SUBAPPLICATION Uebung_016a (* Background Colour umschalten -- 3-fach *)
  (* Standard: 61499-2; Description: Copyright (c) 2023 Meisterschulen am Ostbahnhof This program and the accompanying materials are made available under the terms of the Eclipse Public License 2.0 which is available at https://www.eclipse.org/legal/epl-2.0/ SPDX-License-Identifier: EPL-2.0 *)
  (* Version 1.0, 2023-10-23, Franz Höpfinger, Meisterschulen am Ostbahnhof *)
  IMPORT DefaultPool::SoftKey_F1;
  IMPORT DefaultPool::SoftKey_F2;
  IMPORT DefaultPool::SoftKey_F3;
  IMPORT DefaultPool::SoftKey_F7;
  IMPORT SoftKeyActivationCode::SK_RELEASED;
  IMPORT isobus::ut::colours::COLOR_GREEN;
  IMPORT isobus::ut::colours::COLOR_RED;
  IMPORT isobus::ut::colours::COLOR_WHITE;
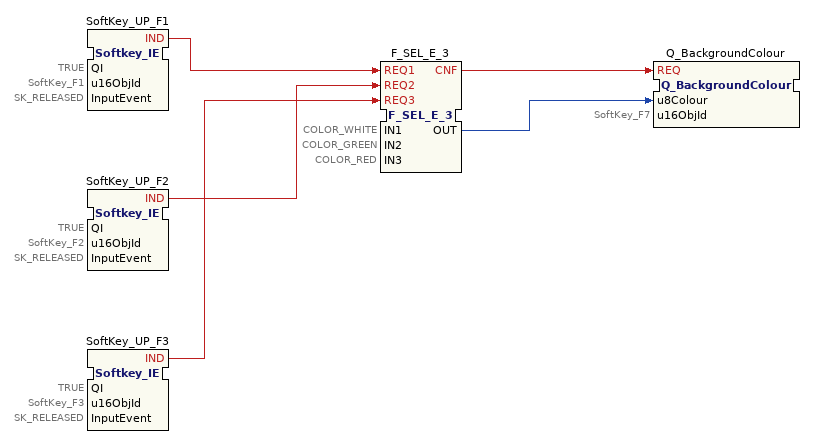
  FBS
    SoftKey_UP_F1 : Softkey_IE(QI := TRUE, u16ObjId := SoftKey_F1, InputEvent := SK_RELEASED);
    SoftKey_UP_F2 : Softkey_IE(QI := TRUE, u16ObjId := SoftKey_F2, InputEvent := SK_RELEASED);
    F_SEL_E_3 : eclipse4diac::utils::selection::F_SEL_E_3(IN1 := COLOR_WHITE, IN2 := COLOR_GREEN, IN3 := COLOR_RED);
    Q_BackgroundColour : isobus::ut::Q_BackgroundColour(u16ObjId := SoftKey_F7);
    SoftKey_UP_F3 : Softkey_IE(QI := TRUE, u16ObjId := SoftKey_F3, InputEvent := SK_RELEASED);
  END_FBS
  EVENT_CONNECTIONS
    F_SEL_E_3.CNF TO Q_BackgroundColour.REQ;
    SoftKey_UP_F1.IND TO F_SEL_E_3.REQ1;
    SoftKey_UP_F2.IND TO F_SEL_E_3.REQ2;
    SoftKey_UP_F3.IND TO F_SEL_E_3.REQ3;
  END_CONNECTIONS
  DATA_CONNECTIONS
    F_SEL_E_3.OUT TO Q_BackgroundColour.u8Colour;
  END_CONNECTIONS
END_SUBAPPLICATION
